// LS Electric XG5000 project: ProjectD
// PLC LSPLC

PROGRAM 컨베이어벨트 (task: 스캔 프로그램)

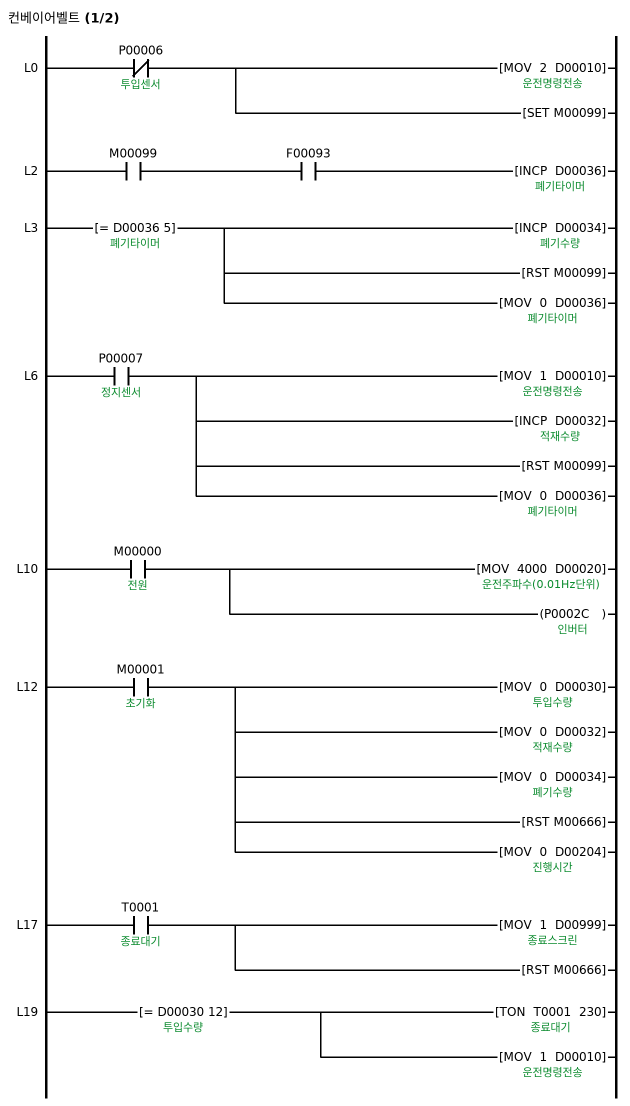
; L0
LOAD NOT  P00006	// 투입센서
MOV       2 D00010	// 운전명령전송
SET       M00099
; L2
LOAD      M00099
AND       F00093
INCP      D00036	// 폐기타이머
; L3
LOAD=     D00036 5	// 폐기타이머
INCP      D00034	// 폐기수량
RST       M00099
MOV       0 D00036	// 폐기타이머
; L6
LOAD      P00007	// 정지센서
MOV       1 D00010	// 운전명령전송
INCP      D00032	// 적재수량
RST       M00099
MOV       0 D00036	// 폐기타이머
; L10
LOAD      M00000	// 전원
MOV       4000 D00020	// 운전주파수(0.01Hz단위)
OUT       P0002C	// 인버터
; L12
LOAD      M00001	// 초기화
MOV       0 D00030	// 투입수량
MOV       0 D00032	// 적재수량
MOV       0 D00034	// 폐기수량
RST       M00666
MOV       0 D00204	// 진행시간
; L17
LOAD      T0001	// 종료대기
MOV       1 D00999	// 종료스크린
RST       M00666
; L19
LOAD=     D00030 12	// 투입수량
TON       T0001 230	// 종료대기
MOV       1 D00010	// 운전명령전송

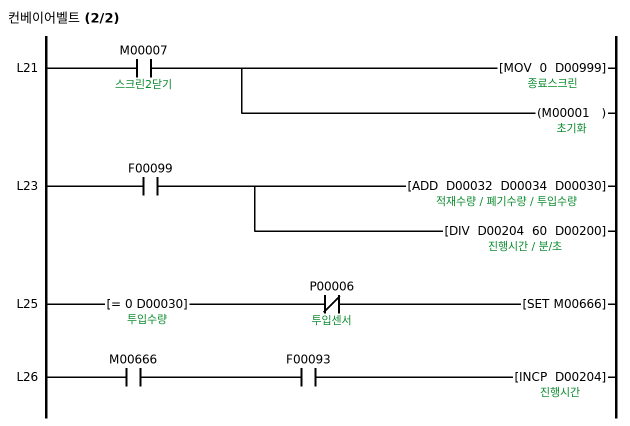
; L21
LOAD      M00007	// 스크린2닫기
MOV       0 D00999	// 종료스크린
OUT       M00001	// 초기화
; L23
LOAD      F00099
ADD       D00032 D00034 D00030	// 적재수량 / 폐기수량 / 투입수량
DIV       D00204 60 D00200	// 진행시간 / 분/초
; L25
LOAD=     0 D00030	// 투입수량
AND NOT   P00006	// 투입센서
SET       M00666
; L26
LOAD      M00666
AND       F00093
INCP      D00204	// 진행시간